// TIA Portal project "Pompe_4" (V15.1)

(* hardware
DEVICE "S71500/ET200MP station_1"  S7-1500 station
   slot 0: "Rail_0"  Rack  6ES7 590-1***0-0AA0
   slot 1: "PLC_1"  CPU 1513-1 PN  6ES7 513-1AL02-0AB0  V2.6
      slot 3: "CPU display_1"  6ES7591-1AA00-0AA0
DEVICE "HMI_1"  KTP900 Basic PN
   slot 0: "HMI_1"  KTP900 Basic PN  6AV2 123-2JB03-0AX0  15.1.0.0
   slot 1: "HMI_RT_1"  KTP900 Basic PN  6AV2 123-2JB03-0AX0  15.1.0.0
   slot 5: "HMI_1.IE_CP_1"  PROFINET Interface  15.0.1.0
      slot 1: "PROFINET Interface_1"  PROFINET Interface
         slot 1: "Port_1"  Port
*)

// ===== PLC "PLC_1"  CPU 1513-1 PN =====

VAR_GLOBAL   // PLC tag table "Default tag table"
   "Clock_Byte" AT %MB0 : Byte;
   "Clock_10Hz" AT %M0.0 : Bool;
   "Clock_5Hz" AT %M0.1 : Bool;
   "Clock_2.5Hz" AT %M0.2 : Bool;
   "Clock_2Hz" AT %M0.3 : Bool;
   "Clock_1.25Hz" AT %M0.4 : Bool;
   "Clock_1Hz" AT %M0.5 : Bool;
   "Clock_0.625Hz" AT %M0.6 : Bool;
   "Clock_0.5Hz" AT %M0.7 : Bool;
END_VAR

VAR_GLOBAL   // PLC tag table "Sistem_1"
   "btn_start_1" AT %I0.0 : Bool;
   "btn_stop_1" AT %I0.1 : Bool;
   "nivel_bazin_1" AT %ID0 : Real;
   "defectiune_sistem_1" AT %I0.2 : Bool;
   "plecare_pompa_1" AT %Q0.0 : Bool;
   "plecare_vana_1" AT %Q0.1 : Bool;
   "indicator_pornit_1" AT %Q0.2 : Bool;
   "mod_1" AT %ID1 : DInt;
END_VAR

VAR_GLOBAL   // PLC tag table "Sistem_2"
   "btn_start_2" AT %I0.3 : Bool;
   "btn_stop_2" AT %I0.4 : Bool;
   "nivel_bazin_2" AT %ID2 : Real;
   "defectiune_sistem_2" AT %I0.5 : Bool;
   "plecare_pompa_2" AT %Q0.3 : Bool;
   "plecare_vana_2" AT %Q0.4 : Bool;
   "indicator_pornit_2" AT %Q0.5 : Bool;
   "mod_2" AT %ID3 : DInt;
END_VAR

VAR_GLOBAL   // PLC tag table "Sistem_3"
   "btn_start_3" AT %I0.6 : Bool;
   "btn_stop_3" AT %I0.7 : Bool;
   "nivel_bazin_3" AT %ID4 : Real;
   "defectiune_sistem_3" AT %I1.0 : Bool;
   "plecare_pompa_3" AT %Q0.6 : Bool;
   "plecare_vana_3" AT %Q0.7 : Bool;
   "indicator_pornit_3" AT %Q1.0 : Bool;
   "mod_3" AT %ID5 : DInt;
END_VAR

VAR_GLOBAL   // PLC tag table "Sistem_4"
   "btn_start_4" AT %I1.1 : Bool;
   "btn_stop_4" AT %I1.2 : Bool;
   "nivel_bazin_4" AT %ID6 : Real;
   "defectiune_sistem_4" AT %I1.3 : Bool;
   "plecare_pompa_4" AT %Q1.1 : Bool;
   "plecare_vana_4" AT %Q1.2 : Bool;
   "indicator_pornit_4" AT %Q1.3 : Bool;
   "mod_4" AT %ID7 : DInt;
END_VAR

DATA_BLOCK "Alarme_DB"   // DB1
{ S7_Optimized_Access := 'TRUE' }
VERSION : 0.1
   VAR
      gather : Word;
      "array" : Array[0..15] of Bool;
   END_VAR
BEGIN
END_DATA_BLOCK

DATA_BLOCK "Avarii_DB"   // DB2
{ S7_Optimized_Access := 'TRUE' }
VERSION : 0.1
   VAR
      esd_1 : Bool;
      btn_esd_1 : Bool;
      reset_esd_1 : Bool;
      avarie_sistem_1 : Bool;
      btn_avarie_sistem_1 : Bool;
      reset_avarie_sistem_1 : Bool;
      esd_2 : Bool;
      btn_esd_2 : Bool;
      reset_esd_2 : Bool;
      btn_avarie_sistem_2 : Bool;
      reset_avarie_sistem_2 : Bool;
      esd_3 : Bool;
      btn_esd_3 : Bool;
      reset_esd_3 : Bool;
      btn_avarie_sistem_3 : Bool;
      reset_avarie_sistem_3 : Bool;
      esd_4 : Bool;
      btn_esd_4 : Bool;
      reset_esd_4 : Bool;
      btn_avarie_sistem_4 : Bool;
      reset_avarie_sistem_4 : Bool;
   END_VAR
BEGIN
END_DATA_BLOCK

DATA_BLOCK "Sistem_1_DB"   // DB3
{ S7_Optimized_Access := 'TRUE' }
VERSION : 0.1
   VAR
      nivel_maxim : Real := 100.0;
      debit_vana : Real := 2.5;
      debit_pompa : Real := 2.5;
      comanda_pornire_pompa : Bool;
      comanda_pornire_vana : Bool;
      permisiune_start : Bool;
      setpoint_pid : Real;
   END_VAR
BEGIN
END_DATA_BLOCK

DATA_BLOCK "Sistem_2_DB"   // DB4
{ S7_Optimized_Access := 'TRUE' }
VERSION : 0.1
BEGIN
END_DATA_BLOCK

DATA_BLOCK "Sistem_3_DB"   // DB5
{ S7_Optimized_Access := 'TRUE' }
VERSION : 0.1
BEGIN
END_DATA_BLOCK

DATA_BLOCK "Sistem_4_DB"   // DB6
{ S7_Optimized_Access := 'TRUE' }
VERSION : 0.1
BEGIN
END_DATA_BLOCK

DATA_BLOCK "Logs_DB"   // DB7
{ S7_Optimized_Access := 'TRUE' }
VERSION : 0.1
BEGIN
END_DATA_BLOCK

DATA_BLOCK "Pompa_sistem_1"   // DB8
{ S7_Optimized_Access := 'TRUE' }
VERSION : 0.1
// stored: InstanceOfName Pompa
"Pompa"
BEGIN
END_DATA_BLOCK

DATA_BLOCK "Vana_sistem_1"   // DB9
{ S7_Optimized_Access := 'TRUE' }
VERSION : 0.1
// stored: InstanceOfName Vana
"Vana"
BEGIN
END_DATA_BLOCK

DATA_BLOCK "Simulare_sistem_1"   // DB14
{ S7_Optimized_Access := 'TRUE' }
VERSION : 0.1
// stored: InstanceOfName Simulare
"Simulare"
BEGIN
END_DATA_BLOCK

DATA_BLOCK "Sistem_1"   // DB15
{ S7_Optimized_Access := 'TRUE' }
VERSION : 0.1
// stored: InstanceOfName Sistem
"Sistem"
BEGIN
END_DATA_BLOCK

// folder: System blocks/Program resources

DATA_BLOCK "timer_reset_pornire_vana"   // DB10
{ S7_Optimized_Access := 'TRUE' }
AUTHOR : Simatic
FAMILY : IEC
NAME : IEC_TMR
VERSION : 1.0
// stored: InstanceOfName IEC_TIMER
"IEC_TIMER"
BEGIN
END_DATA_BLOCK

DATA_BLOCK "timer_reset_pornire_pompa"   // DB11
{ S7_Optimized_Access := 'TRUE' }
AUTHOR : Simatic
FAMILY : IEC
NAME : IEC_TMR
VERSION : 1.0
// stored: InstanceOfName IEC_TIMER
"IEC_TIMER"
BEGIN
END_DATA_BLOCK

// folder: (top level)

FUNCTION_BLOCK "Sistem"   // FB1, LAD
{ S7_Optimized_Access := 'TRUE' }
VERSION : 0.1
   VAR_INPUT
      nivel_maxim : Real;
      debit_vana : Real;
      debit_pompa : Real;
      "mod" : DInt;
   END_VAR
   VAR_OUTPUT
      comanda_pompa_pornita : Bool;
      comanda_vana_pornita : Bool;
      alarma_sistem : Bool;
      alarma_esd : Bool;
      esd : Bool;
      avarie_sistem : Bool;
      permisiune_start : Bool;
      "status_pornit(HMI)" : Bool;
   END_VAR
   VAR_IN_OUT
      comanda_start : Bool;
      comanda_stop : Bool;
      comanda_pornire_pompa : Bool;
      comanda_pornire_vana : Bool;
      nivel_curent : Real;
      btn_esd : Bool;
      reset_esd : Bool;
      btn_avarie_sistem : Bool;
      reset_avarie_sistem : Bool;
   END_VAR
   VAR
      status_pornit_pompa : Bool;
      status_pornit_vana : Bool;
      resetare_comanda_vana : Bool;
      resetare_comanda_pompa : Bool;
      timer_reset_esd : TON_TIME;
      timer_reset_avarie_sistem : TON_TIME;
      timer_reset_comanda_stop : TON_TIME;
   END_VAR
   VAR_TEMP   // added for the SCL form of the ladder/FBD networks
      _w1 : Bool;
      _w2 : Bool;
   END_VAR
BEGIN

REGION Network 1: comanda buton start
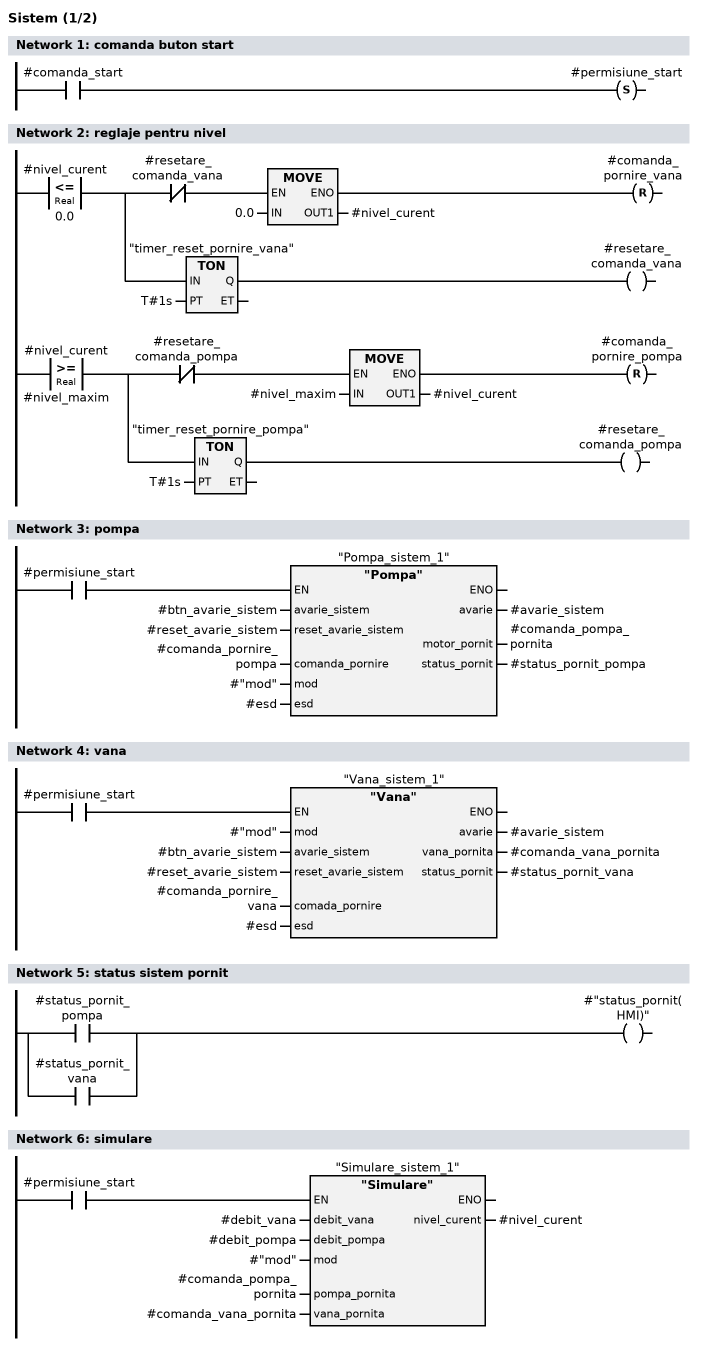
   RUNG wire#powerrail
      Contact( #comanda_start )
      S_Coil( #permisiune_start )
   END_RUNG
   // the same network as SCL:
   IF #comanda_start THEN #permisiune_start := TRUE; END_IF;
END_REGION

REGION Network 2: reglaje pentru nivel
   #_w1 := #nivel_curent <= 0.0;
   IF #_w1 AND NOT #resetare_comanda_vana THEN
       #nivel_curent := 0.0;
       #comanda_pornire_vana := FALSE;
   END_IF;
   "timer_reset_pornire_vana".TON(IN := #_w1, PT := T#1s);
   #resetare_comanda_vana := "timer_reset_pornire_vana".Q;
   #_w2 := #nivel_curent >= #nivel_maxim;
   IF #_w2 AND NOT #resetare_comanda_pompa THEN
       #nivel_curent := #nivel_maxim;
       #comanda_pornire_pompa := FALSE;
   END_IF;
   "timer_reset_pornire_pompa".TON(IN := #_w2, PT := T#1s);
   #resetare_comanda_pompa := "timer_reset_pornire_pompa".Q;
END_REGION

REGION Network 3: pompa
   RUNG wire#powerrail
      Contact( #permisiune_start )
      "Pompa_sistem_1"(avarie_sistem := #btn_avarie_sistem, reset_avarie_sistem := #reset_avarie_sistem, comanda_pornire := #comanda_pornire_pompa, "mod" := #"mod", esd := #esd, avarie => #avarie_sistem, motor_pornit => #comanda_pompa_pornita, status_pornit => #status_pornit_pompa)
   END_RUNG
   // the same network as SCL:
   IF #permisiune_start THEN
       "Pompa_sistem_1"(avarie_sistem := #btn_avarie_sistem,   // "Pompa"
                        reset_avarie_sistem := #reset_avarie_sistem,
                        comanda_pornire := #comanda_pornire_pompa,
                        "mod" := #"mod",
                        esd := #esd,
                        avarie => #avarie_sistem,
                        motor_pornit => #comanda_pompa_pornita,
                        status_pornit => #status_pornit_pompa);
   END_IF;
END_REGION

REGION Network 4: vana
   RUNG wire#powerrail
      Contact( #permisiune_start )
      "Vana_sistem_1"("mod" := #"mod", avarie_sistem := #btn_avarie_sistem, reset_avarie_sistem := #reset_avarie_sistem, comada_pornire := #comanda_pornire_vana, esd := #esd, avarie => #avarie_sistem, vana_pornita => #comanda_vana_pornita, status_pornit => #status_pornit_vana)
   END_RUNG
   // the same network as SCL:
   IF #permisiune_start THEN
       "Vana_sistem_1"("mod" := #"mod",   // "Vana"
                       avarie_sistem := #btn_avarie_sistem,
                       reset_avarie_sistem := #reset_avarie_sistem,
                       comada_pornire := #comanda_pornire_vana,
                       esd := #esd,
                       avarie => #avarie_sistem,
                       vana_pornita => #comanda_vana_pornita,
                       status_pornit => #status_pornit_vana);
   END_IF;
END_REGION

REGION Network 5: status sistem pornit
   RUNG wire#powerrail
      Contact( #status_pornit_pompa )
      wire#w1
      Coil( #"status_pornit(HMI)" )
   END_RUNG
   RUNG wire#powerrail
      Contact( #status_pornit_vana )
   END_RUNG wire#w1
   // the same network as SCL:
   #"status_pornit(HMI)" := #status_pornit_pompa OR #status_pornit_vana;
END_REGION

REGION Network 6: simulare
   RUNG wire#powerrail
      Contact( #permisiune_start )
      "Simulare_sistem_1"(debit_vana := #debit_vana, debit_pompa := #debit_pompa, "mod" := #"mod", pompa_pornita := #comanda_pompa_pornita, vana_pornita := #comanda_vana_pornita, nivel_curent => #nivel_curent)
   END_RUNG
   // the same network as SCL:
   IF #permisiune_start THEN
       "Simulare_sistem_1"(debit_vana := #debit_vana,   // "Simulare"
                           debit_pompa := #debit_pompa,
                           "mod" := #"mod",
                           pompa_pornita := #comanda_pompa_pornita,
                           vana_pornita := #comanda_vana_pornita,
                           nivel_curent => #nivel_curent);
   END_IF;
END_REGION

REGION Network 7: esd
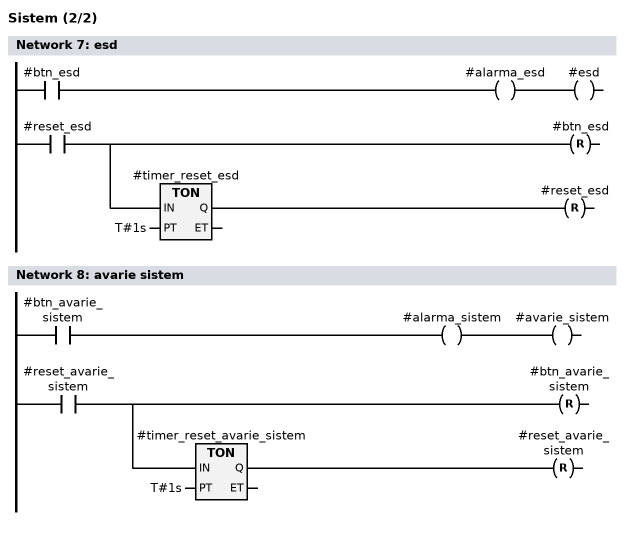
   #alarma_esd := #btn_esd;
   #esd := #btn_esd;
   IF #reset_esd THEN #btn_esd := FALSE; END_IF;
   #timer_reset_esd(IN := #reset_esd, PT := T#1s);   // TON
   IF #timer_reset_esd.Q THEN #reset_esd := FALSE; END_IF;
END_REGION

REGION Network 8: avarie sistem
   #alarma_sistem := #btn_avarie_sistem;
   #avarie_sistem := #btn_avarie_sistem;
   IF #reset_avarie_sistem THEN #btn_avarie_sistem := FALSE; END_IF;
   #timer_reset_avarie_sistem(IN := #reset_avarie_sistem, PT := T#1s);   // TON
   IF #timer_reset_avarie_sistem.Q THEN #reset_avarie_sistem := FALSE; END_IF;
END_REGION
END_FUNCTION_BLOCK

FUNCTION_BLOCK "Pompa"   // FB2, LAD
{ S7_Optimized_Access := 'TRUE' }
VERSION : 0.1
   VAR_INPUT
      avarie_sistem : Bool;
      reset_avarie_sistem : Bool;
      comanda_pornire : Bool;
      "mod" : DInt;
      esd : Bool;
   END_VAR
   VAR_OUTPUT
      avarie : Bool;
      motor_pornit : Bool;
      status_pornit : Bool;
   END_VAR
BEGIN

REGION Network 1: pornire pompa pe oricem od de functionare
   // 0 - manual, 1 - auto
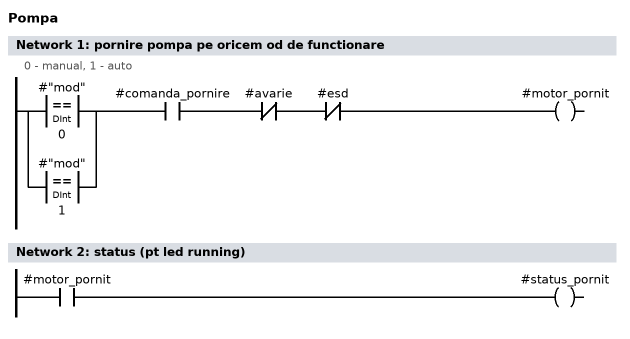
   RUNG wire#powerrail
      { S7_Templates := "SrcType := DInt" } EQ_Contact(in1 := #"mod", in2 := 0)
      wire#w1
      Contact( #comanda_pornire )
      I_Contact( #avarie )
      I_Contact( #esd )
      Coil( #motor_pornit )
   END_RUNG
   RUNG wire#powerrail
      { S7_Templates := "SrcType := DInt" } EQ_Contact(in1 := #"mod", in2 := 1)
   END_RUNG wire#w1
   // the same network as SCL:
   #motor_pornit := ((#"mod" = 0) OR (#"mod" = 1)) AND #comanda_pornire AND NOT #avarie AND NOT #esd;
END_REGION

REGION Network 2: status (pt led running)
   RUNG wire#powerrail
      Contact( #motor_pornit )
      Coil( #status_pornit )
   END_RUNG
   // the same network as SCL:
   #status_pornit := #motor_pornit;
END_REGION
END_FUNCTION_BLOCK

FUNCTION_BLOCK "Vana"   // FB3, LAD
{ S7_Optimized_Access := 'TRUE' }
VERSION : 0.1
   VAR_INPUT
      "mod" : DInt;
      avarie_sistem : Bool;
      reset_avarie_sistem : Bool;
      comada_pornire : Bool;
      esd : Bool;
   END_VAR
   VAR_OUTPUT
      avarie : Bool;
      vana_pornita : Bool;
      status_pornit : Bool;
   END_VAR
BEGIN

REGION Network 1: pornire pompa pe oricem od de functionare
   // 0 - manual, 1 - auto
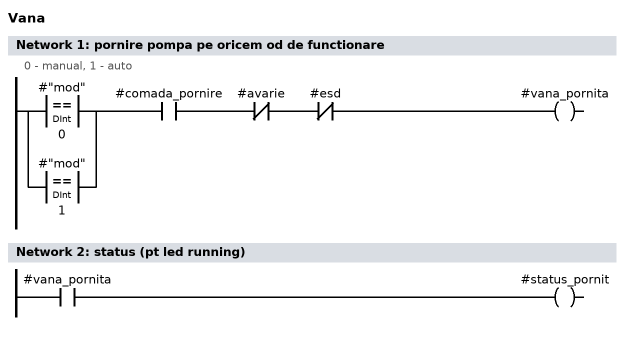
   RUNG wire#powerrail
      { S7_Templates := "SrcType := DInt" } EQ_Contact(in1 := #"mod", in2 := 0)
      wire#w1
      Contact( #comada_pornire )
      I_Contact( #avarie )
      I_Contact( #esd )
      Coil( #vana_pornita )
   END_RUNG
   RUNG wire#powerrail
      { S7_Templates := "SrcType := DInt" } EQ_Contact(in1 := #"mod", in2 := 1)
   END_RUNG wire#w1
   // the same network as SCL:
   #vana_pornita := ((#"mod" = 0) OR (#"mod" = 1)) AND #comada_pornire AND NOT #avarie AND NOT #esd;
END_REGION

REGION Network 2: status (pt led running)
   RUNG wire#powerrail
      Contact( #vana_pornita )
      Coil( #status_pornit )
   END_RUNG
   // the same network as SCL:
   #status_pornit := #vana_pornita;
END_REGION
END_FUNCTION_BLOCK

FUNCTION_BLOCK "Simulare"   // FB4, LAD
{ S7_Optimized_Access := 'TRUE' }
VERSION : 0.1
   VAR_INPUT
      debit_vana : Real;
      debit_pompa : Real;
      "mod" : DInt;
      pompa_pornita : Bool;
      vana_pornita : Bool;
   END_VAR
   VAR_OUTPUT
      nivel_curent : Real;
   END_VAR
   VAR
      re1 : Bool;
      re2 : Bool;
   END_VAR
   VAR_TEMP   // added for the SCL form of the ladder/FBD networks
      _w1 : Bool;
   END_VAR
BEGIN

REGION Network 1: umple cu pompa
   // asta pe mod 0 manual, pe auto, o sa fie bloc separat cu pid
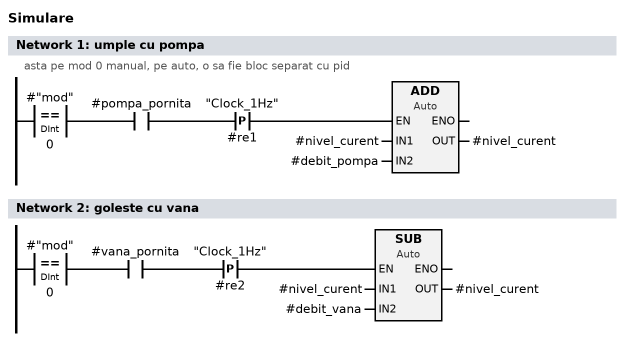
   RUNG wire#powerrail
      { S7_Templates := "SrcType := DInt" } EQ_Contact(in1 := #"mod", in2 := 0)
      Contact( #pompa_pornita )
      P_Contact(operand := "Clock_1Hz", bit := #re1)
      Add(in1 := #nivel_curent, in2 := #debit_pompa, out => #nivel_curent)
   END_RUNG
   // the same network as SCL:
   #_w1 := (#"mod" = 0) AND #pompa_pornita AND "Clock_1Hz" AND NOT #re1;   // rising edge of "Clock_1Hz"
   #re1 := "Clock_1Hz";
   IF #_w1 THEN #nivel_curent := #nivel_curent + #debit_pompa; END_IF;
END_REGION

REGION Network 2: goleste cu vana
   RUNG wire#powerrail
      { S7_Templates := "SrcType := DInt" } EQ_Contact(in1 := #"mod", in2 := 0)
      Contact( #vana_pornita )
      P_Contact(operand := "Clock_1Hz", bit := #re2)
      Sub(in1 := #nivel_curent, in2 := #debit_vana, out => #nivel_curent)
   END_RUNG
   // the same network as SCL:
   #_w1 := (#"mod" = 0) AND #vana_pornita AND "Clock_1Hz" AND NOT #re2;   // rising edge of "Clock_1Hz"
   #re2 := "Clock_1Hz";
   IF #_w1 THEN #nivel_curent := #nivel_curent - #debit_vana; END_IF;
END_REGION
END_FUNCTION_BLOCK

ORGANIZATION_BLOCK "Main"   // OB1, LAD, ProgramCycle
TITLE = "Main Program Sweep (Cycle)"
{ S7_Optimized_Access := 'TRUE' }
VERSION : 0.1
   VAR_INPUT
      Initial_Call : Bool;   // Initial call of this OB
      Remanence : Bool;   // =True, if remanent data are available
   END_VAR
BEGIN

REGION Network 1: Gather pe alarme
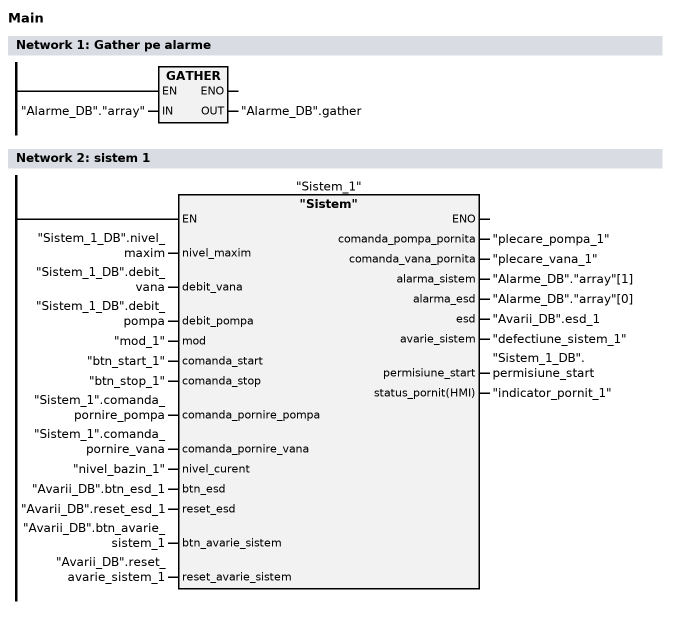
   GATHER(IN := "Alarme_DB"."array", OUT => "Alarme_DB".gather);
END_REGION

REGION Network 2: sistem 1
   RUNG wire#powerrail
      "Sistem_1"(nivel_maxim := "Sistem_1_DB".nivel_maxim, debit_vana := "Sistem_1_DB".debit_vana, debit_pompa := "Sistem_1_DB".debit_pompa, "mod" := "mod_1", comanda_start := "btn_start_1", comanda_stop := "btn_stop_1", comanda_pornire_pompa := "Sistem_1".comanda_pornire_pompa, comanda_pornire_vana := "Sistem_1".comanda_pornire_vana, nivel_curent := "nivel_bazin_1", btn_esd := "Avarii_DB".btn_esd_1, reset_esd := "Avarii_DB".reset_esd_1, btn_avarie_sistem := "Avarii_DB".btn_avarie_sistem_1, reset_avarie_sistem := "Avarii_DB".reset_avarie_sistem_1, comanda_pompa_pornita => "plecare_pompa_1", comanda_vana_pornita => "plecare_vana_1", alarma_sistem => "Alarme_DB"."array"[1], alarma_esd => "Alarme_DB"."array"[0], esd => "Avarii_DB".esd_1, avarie_sistem => "defectiune_sistem_1", permisiune_start => "Sistem_1_DB".permisiune_start, "status_pornit(HMI)" => "indicator_pornit_1")
   END_RUNG
   // the same network as SCL:
   "Sistem_1"(nivel_maxim := "Sistem_1_DB".nivel_maxim,   // "Sistem"
              debit_vana := "Sistem_1_DB".debit_vana,
              debit_pompa := "Sistem_1_DB".debit_pompa,
              "mod" := "mod_1",
              comanda_start := "btn_start_1",
              comanda_stop := "btn_stop_1",
              comanda_pornire_pompa := "Sistem_1".comanda_pornire_pompa,
              comanda_pornire_vana := "Sistem_1".comanda_pornire_vana,
              nivel_curent := "nivel_bazin_1",
              btn_esd := "Avarii_DB".btn_esd_1,
              reset_esd := "Avarii_DB".reset_esd_1,
              btn_avarie_sistem := "Avarii_DB".btn_avarie_sistem_1,
              reset_avarie_sistem := "Avarii_DB".reset_avarie_sistem_1,
              comanda_pompa_pornita => "plecare_pompa_1",
              comanda_vana_pornita => "plecare_vana_1",
              alarma_sistem => "Alarme_DB"."array"[1],
              alarma_esd => "Alarme_DB"."array"[0],
              esd => "Avarii_DB".esd_1,
              avarie_sistem => "defectiune_sistem_1",
              permisiune_start => "Sistem_1_DB".permisiune_start,
              "status_pornit(HMI)" => "indicator_pornit_1");
END_REGION
END_ORGANIZATION_BLOCK

(* ===== HMI "HMI_RT_1" =====
system functions are stored by id; their names below are inferred from use
connection "HMI_Connection_1": ETHERNET, SMART_S7_1500_OMS

HMI tags "Default tag table"
   "Alarme_DB_gather" : Word = PLC Alarme_DB.gather, 1 s
   "Avarii_DB_esd_1" : Bool = PLC Avarii_DB.esd_1, 1 s
   "defectiune_sistem_1" : Bool = PLC defectiune_sistem_1 AT %I0.2, 1 s
   "Sistem_1_status_pornit(HMI)" : Bool = PLC Sistem_1.status_pornit(HMI), 1 s
   "indicator_pornit_1" : Bool = PLC indicator_pornit_1 AT %Q0.2, 1 s
   "Avarii_DB_btn_esd_1" : Bool = PLC Avarii_DB.btn_esd_1, 1 s
   "Avarii_DB_reset_esd_1" : Bool = PLC Avarii_DB.reset_esd_1, 1 s
   "Avarii_DB_btn_avarie_sistem_1" : Bool = PLC Avarii_DB.btn_avarie_sistem_1, 1 s
   "Avarii_DB_reset_avarie_sistem_1" : Bool = PLC Avarii_DB.reset_avarie_sistem_1, 1 s
   "btn_start_1" : Bool = PLC btn_start_1 AT %I0.0, 1 s
   "btn_stop_1" : Bool = PLC btn_stop_1 AT %I0.1, 1 s
   "nivel_bazin_1" : Real = PLC nivel_bazin_1 AT %ID0, 1 s
   "Sistem_1_mod" : DInt = PLC Sistem_1.mod, 1 s
   "mod_1" : DInt = PLC mod_1 AT %ID1, 1 s
   "Sistem_1_DB_setpoint_pid" : Real = PLC Sistem_1_DB.setpoint_pid, 1 s
   "plecare_pompa_1" : Bool = PLC plecare_pompa_1 AT %Q0.0, 1 s
   "plecare_vana_1" : Bool = PLC plecare_vana_1 AT %Q0.1, 1 s
   "Sistem_1_DB_permisiune_start" : Bool = PLC Sistem_1_DB.permisiune_start, 1 s

discrete alarms
   1: 'ESD', class Errors, trigger "Alarme_DB_gather" bit 0
   2: 'Avarie sistem', class Errors, trigger "Alarme_DB_gather" bit 1

text list "Moduri": 0 'Manual'; 1 'Automat'

Template "Template_1" 800x480
   Button "Exit" at 722,440 size 55x39; TextOff 'Exit'; PictureOff "ExitRuntime_KTP900_Basic_PN_TR"; PictureOn "ExitRuntime_KTP900_Basic_PN_TR"
      on Release: StopRuntime(0)

screen "Pompa1" 800x480, template "Template_1"
   TextField "Text field_1" at 23,455 size 60x20; Text 'Pompa 1'
   TextField "Text field_2" at 121,455 size 60x20; Text 'Pompa 2'
   TextField "Text field_3" at 221,455 size 60x20; Text 'Pompa 3'
   TextField "Text field_4" at 321,455 size 60x20; Text 'Pompa 4'
   TextField "Text field_5" at 431,455 size 35x20; Text 'Logs'
   TrendView "Trend view_1" at 0,217 size 800x225
   Bar "Bar_1" at 582,56 size 165x149; MinimumValue 0; MaximumValue 100
      ProcessValue <- "nivel_bazin_1"
   IOField "I/O field_1" at 618,24 size 96x32; FormatPattern 999.99; Unit L
      ProcessValue <- "nivel_bazin_1"
   TextField "Text field_6" at 357,3 size 88x27; Text 'Pompa 1'
   TextField "Text field_7" at 646,4 size 39x20; Text 'Bazin'
   Button "Button_1" at 26,115 size 55x32; TextOff 'ESD'
      on Click: SetBit("Avarii_DB_btn_esd_1")
   Button "Button_2" at 26,147 size 55x32; TextOff 'Reset'
      on Click: SetBit("Avarii_DB_reset_esd_1")
   Circle "Circle_1" at 30,55 size 48x48
      Appearance <- "Avarii_DB_esd_1"
   SymbolicIOField "Symbolic I/O field_1" at 351,73 size 101x32; TextOff '0'; TextOn '1'; TextList "Moduri"
      ProcessValue <- "mod_1"
   Button "Button_3" at 105,115 size 55x32; TextOff 'Avarie'
      on Click: SetBit("Avarii_DB_btn_avarie_sistem_1")
   Button "Button_4" at 105,147 size 55x32; TextOff 'Reset'
      on Click: SetBit("Avarii_DB_reset_avarie_sistem_1")
   Circle "Circle_2" at 109,55 size 48x48
      Appearance <- "defectiune_sistem_1"
   IOField "I/O field_2" at 351,135 size 101x32; FormatPattern 999.99; Unit L
      Visibility <- "mod_1"
      ProcessValue <- "Sistem_1_DB_setpoint_pid"
   TextField "Text field_8" at 383,52 size 32x20; Text 'Mod'
   TextField "Text field_9" at 358,115 size 86x20; Text 'Setpoint PID'
      Visibility <- "mod_1"
   Button "Button_5" at 480,75 size 27x28; TextOff 'On'
      Visibility <- "mod_1"
      on Click: SetTag("plecare_pompa_1", 1)
   Button "Button_6" at 511,75 size 27x28; TextOff 'Off'
      Visibility <- "mod_1"
      on Click: SetTag("plecare_pompa_1", 0)
   TextField "Text field_10" at 485,54 size 48x20; Text 'Pompa'
      Visibility <- "mod_1"
   Button "Button_7" at 480,126 size 27x28; TextOff 'On'
      Visibility <- "mod_1"
      on Click: SetTag("plecare_vana_1", 1)
   Button "Button_8" at 511,126 size 27x28; TextOff 'Off'
      Visibility <- "mod_1"
      on Click: SetTag("plecare_vana_1", 0)
   TextField "Text field_11" at 489,105 size 38x20; Text 'Vana'
      Visibility <- "mod_1"
   Circle "Circle_3" at 189,55 size 48x48
      Appearance <- "Sistem_1_DB_permisiune_start"
   TextField "Text field_13" at 275,59 size 44x20; Text 'Pornit'
   Button "Button_9" at 189,115 size 46x32; TextOff 'Start'
      on Click: SetBit("btn_start_1")
   Button "Button_10" at 189,147 size 46x32; TextOff 'Stop'
      on Click: SetBit("btn_stop_1")
   Circle "Circle_4" at 267,88 size 61x61
      Appearance <- "indicator_pornit_1"

screen "Pompa2" 800x480
   TextField "Text field_1" at 23,455 size 60x20; Text 'Pompa 1'
   TextField "Text field_2" at 121,455 size 60x20; Text 'Pompa 2'
   TextField "Text field_3" at 221,455 size 60x20; Text 'Pompa 3'
   TextField "Text field_4" at 321,455 size 60x20; Text 'Pompa 4'
   TextField "Text field_5" at 431,455 size 35x20; Text 'Logs'

screen "Pompa3" 800x480
   TextField "Text field_1" at 23,455 size 60x20; Text 'Pompa 1'
   TextField "Text field_2" at 121,455 size 60x20; Text 'Pompa 2'
   TextField "Text field_3" at 221,455 size 60x20; Text 'Pompa 3'
   TextField "Text field_4" at 321,455 size 60x20; Text 'Pompa 4'
   TextField "Text field_5" at 431,455 size 35x20; Text 'Logs'

screen "Pompa4" 800x480
   TextField "Text field_1" at 23,455 size 60x20; Text 'Pompa 1'
   TextField "Text field_2" at 121,455 size 60x20; Text 'Pompa 2'
   TextField "Text field_3" at 221,455 size 60x20; Text 'Pompa 3'
   TextField "Text field_4" at 321,455 size 60x20; Text 'Pompa 4'
   TextField "Text field_5" at 431,455 size 35x20; Text 'Logs'

screen "Logs" 800x480
   TextField "Text field_1" at 23,455 size 60x20; Text 'Pompa 1'
   TextField "Text field_2" at 121,455 size 60x20; Text 'Pompa 2'
   TextField "Text field_3" at 221,455 size 60x20; Text 'Pompa 3'
   TextField "Text field_4" at 321,455 size 60x20; Text 'Pompa 4'
   TextField "Text field_5" at 431,455 size 35x20; Text 'Logs'
*)